PROGRAM MAIN
VAR
	brakes AT %Q*: BYTE;
END_VAR

END_PROGRAM

(* stored: Version 1.1.0.1, ProductVersion 3.1.4020.12
   POU MAIN: Id {64193399-6c38-4426-a728-06ada0c3f571}, SpecialFunc None *)
